(* CODESYS project Cooling System.project
   Title: Cooling System
   Version: 0.0.0.0
   Author: Admin

Project tree, tasks and I/O mapping:
  MyController : TM241CE40T/U, Schneider Electric, order no. TM241CE40T/U, version 4.0.5.9
    application Application
      task MAST (cyclic, interval 20 ms, priority 15, watchdog 100 ms x 1) calls Main
      SUBPROGRAM/
        HMIdriver/
        IOdriver/
          program IOinput [ST]
          program IOoutput [ST]
          function AnalogValue [ST]
      VAR/
        global variables GVL
        global variables GVL_IO
    DI : Digital Inputs, Schneider Electric, version 4.0.5.9
        input  idwDI_IDW0 : DWORD  // IDW0
        input  ibDI_IB1 : BYTE  // IB1
    DQ : Digital Outputs, Schneider Electric, version 4.0.5.9
        output qwDQ_QW0 : WORD  // QW0
        output qbDQ_QB1 : BYTE  // QB1
    Counters : Counters, Schneider Electric, version 4.0.5.9
    Pulse_Generators : Pulse Generators, Schneider Electric, version 4.0.5.9
    Cartridge_1 : Cartridge, Schneider Electric, version 4.0.5.9
    Cartridge_2 : Cartridge, Schneider Electric, version 4.0.5.9
    IO_Bus : IO bus - TM3, Schneider Electric, version 4.0.5.9
      AIModule_1 : TM3AI8/G, Schneider Electric, order no. TM3AI8/G, version 1.0.0.16
          input  iiModule_1_IW0 : INT  // IW0
          input  iiModule_1_IW1 : INT  // IW1
          input  iiModule_1_IW2 : INT  // IW2
          input  iiModule_1_IW3 : INT  // IW3
          input  iiModule_1_IW4 : INT  // IW4
          input  iiModule_1_IW5 : INT  // IW5
          input  iiModule_1_IW6 : INT  // IW6
          input  iiModule_1_IW7 : INT  // IW7
          input  ibModule_1_IBStatusIW0 : BYTE  // IBStatusIW0
          input  ibModule_1_IBStatusIW1 : BYTE  // IBStatusIW1
          input  ibModule_1_IBStatusIW2 : BYTE  // IBStatusIW2
          input  ibModule_1_IBStatusIW3 : BYTE  // IBStatusIW3
          input  ibModule_1_IBStatusIW4 : BYTE  // IBStatusIW4
          input  ibModule_1_IBStatusIW5 : BYTE  // IBStatusIW5
          input  ibModule_1_IBStatusIW6 : BYTE  // IBStatusIW6
          input  ibModule_1_IBStatusIW7 : BYTE  // IBStatusIW7
      TIModule_2 : TM3TI4/G, Schneider Electric, order no. TM3TI4/G, version 1.0.1.4
          input  iiModule_2_IW0 : INT  // IW0
          input  iiModule_2_IW1 : INT  // IW1
          input  iiModule_2_IW2 : INT  // IW2
          input  iiModule_2_IW3 : INT  // IW3
          input  ibModule_2_IBStatusIW0 : BYTE  // IBStatusIW0
          input  ibModule_2_IBStatusIW1 : BYTE  // IBStatusIW1
          input  ibModule_2_IBStatusIW2 : BYTE  // IBStatusIW2
          input  ibModule_2_IBStatusIW3 : BYTE  // IBStatusIW3
    COM_Bus : COM bus, Schneider Electric, version 4.0.5.9
    Ethernet_1 : Ethernet Network, Schneider Electric, version 4.0.5.9
    Serial_Line_1 : Serial line, Schneider Electric, version 4.0.5.9
      SoMachine_Network_Manager : SoMachine-Network Manager, Schneider Electric, version 4.0.0.2
    Serial_Line_2 : Serial line, Schneider Electric, version 4.0.5.9
      Modbus_Manager : Modbus Manager, Schneider Electric, version 4.0.0.2
  FdtConnections : FDT Connections, Schneider Electric, version 1.0.0.2
  program Main [ST]
*)

// MyController/Application/VAR/GVL
VAR_GLOBAL
END_VAR

// MyController/Application/VAR/GVL_IO
VAR_GLOBAL
//----- Инверсии входов-выходов -----
	InvDI1_PLC	AT %MW220: WORD;	// Входы ПЛК
	InvDI2_PLC	AT %MW221: WORD;	// Входы ПЛК

	InvDO_PLC	AT %MW230: WORD;	// Выходы ПЛК
	
//----- ОБЪЯВЛЕНИЕ ПОРТОВ -----
	PortDI1_PLC	AT %MW200: WORD;
	PortDI2_PLC	AT %MW201: WORD;
	
	PortDO_PLC	AT %MW210: WORD;

//----- ДИСКРЕТНЫЕ ВХОДЫ -----
	sbReset		: BOOL;		// SB17 - Сброс кнопка

//----- ДИСКРЕТНЫЕ ВЫХОДЫ -----	
	hlFault		: BOOL;		// HL31 - Авария

END_VAR

// Main
PROGRAM Main
VAR
END_VAR

IOinput();





IOoutput();

END_PROGRAM

// MyController/Application/SUBPROGRAM/IOdriver/IOinput
PROGRAM IOinput
VAR
END_VAR

//***** Дискретные входы *****
// Инверсия входов
// Приходится делать побитово для облегчения перетаскивания тегов в панель визуализации

PortDI1_PLC := InvDI1_PLC XOR DWORD_TO_WORD(idwDI_IDW0) ;
PortDI2_PLC := InvDI2_PLC XOR DWORD_TO_WORD(SHR(idwDI_IDW0,8)) ;

// ***** Привязка дискретных входов *****
// Входы ПЛК
sbReset		:= PortDI1_PLC.0; 			// Кнопка Квитирование защит

END_PROGRAM

// MyController/Application/SUBPROGRAM/IOdriver/IOoutput
PROGRAM IOoutput
VAR
END_VAR

//***** Привязка и инверсия дискретных выходов *****

//Выходы PLC
{ PortDO_PLC.0		:= hlReset 					XOR InvDO_PLC.0;	// SB17 - кнопка Сброс защит
PortDO_PLC.1		:= hlReady					XOR	InvDO_PLC.1;
PortDO_PLC.2		:= hlFault					XOR InvDO_PLC.2;
PortDO_PLC.3		:= hlLamp					XOR InvDO_PLC.3;
PortDO_PLC.4		:= InvDO_PLC.4;
PortDO_PLC.5		:= InvDO_PLC.5;
PortDO_PLC.6		:= InvDO_PLC.6;
PortDO_PLC.7		:= InvDO_PLC.7;
PortDO_PLC.8		:= kBanPump1				XOR InvDO_PLC.8;	// Запрет включения Насос 1 (К33)
PortDO_PLC.9		:= kBanPump2				XOR InvDO_PLC.9;	// Запрет включения Насос 2 (К34)
}
// Перекладываем сформированные сигналы в выходные модули
qwDQ_QW0		:= PortDO_PLC;

END_PROGRAM

// MyController/Application/SUBPROGRAM/IOdriver/AnalogValue
FUNCTION AnalogValue : REAL
VAR_INPUT
	IN		: INT;	// Входное значение
	OFFSET	: INT;	// Смещение нуля (значение * 100)
END_VAR
VAR
	Val		: REAL;	// Значение напряжения на входе
END_VAR

// Вход 10..+10В = -32768...32767 дискрет
// В вольтах напряжение на входе = (IN/32767) * 10В
Val := (INT_TO_REAL(IN)/32767.0)*10.0; 

AnalogValue := Val + INT_TO_REAL(OFFSET)/100.0;

END_FUNCTION
